(* IEC 61131-3 sources: SmartHomeNew/snapshots/2026-05-07 (part 2) *)

(* ---- FB_Modbus_RTU_SysCom_Backend.st ---- *)
FUNCTION_BLOCK FB_Modbus_RTU_SysCom_Backend
VAR_INPUT
    VI_Enable : BOOL;
    VI_System_Time_MS : UDINT;
END_VAR

VAR
    L_Result : UDINT;
    L_Handle : UDINT := 16#FFFFFFFF;

    L_Settings : SysCom.SysComSettings;
    L_SettingsEx2 : SysCom.SysComSettingsEx2;

    L_Bytes_Written : UDINT;
    L_Bytes_Read : UDINT;

    L_RX_Buffer : ARRAY[0..255] OF BYTE;

    L_Open_Done : BOOL := FALSE;
    L_i : INT;
    L_j : INT;
    L_Read_Count : INT;
    L_Target_Index : INT;
    L_Frame_Length : INT;

    L_CRC : WORD;
    L_CRC_Frame : WORD;

    L_Baudrate : UDINT;
    L_Interframe_MS : UDINT;
END_VAR

// ======================================================
// MODBUS RTU SYSCOM BACKEND
// ======================================================
// Industrial transport runtime:
//   - serial open/configure
//   - RX assembler
//   - CRC validation
//   - watchdog supervision
//   - reconnect supervision
// ======================================================

IF NOT VI_Enable THEN

    IF L_Handle <> 16#FFFFFFFF THEN
        SysCom.SysComClose(hCom := L_Handle);
        L_Handle := 16#FFFFFFFF;
    END_IF;

    L_Open_Done := FALSE;

    GVL_MODBUS_SYSCOM_TRANSPORT.G_Transport_Attached := FALSE;
    GVL_MODBUS_SYSCOM_TRANSPORT.G_Backend_Online := FALSE;

    GVL_MODBUS_SYSCOM_TRANSPORT.G_Backend_State :=
        MB_SYSCOM_CLOSED;

    GVL_MODBUS_SYSCOM_TRANSPORT.G_RX_State :=
        MB_RTU_RX_IDLE;

    GVL_MODBUS_SYSCOM_TRANSPORT.G_RX_Assembler_Active := FALSE;
    GVL_MODBUS_SYSCOM_TRANSPORT.G_RX_Assembler_Length := 0;

    RETURN;
END_IF;

// ======================================================
// WATCHDOGS
// ======================================================
GVL_MODBUS_SYSCOM_TRANSPORT.G_TX_Watchdog_Timeout := FALSE;
GVL_MODBUS_SYSCOM_TRANSPORT.G_RX_Watchdog_Timeout := FALSE;
GVL_MODBUS_SYSCOM_TRANSPORT.G_Bus_Silent := FALSE;

IF GVL_MODBUS_SYSCOM_TRANSPORT.G_TX_Request THEN

    IF (VI_System_Time_MS -
        GVL_MODBUS_SYSCOM_TRANSPORT.G_Last_TX_Request_MS) >
        (GVL_CONFIG.G_Modbus_RTU_Request_Timeout_MS * 2) THEN

        GVL_MODBUS_SYSCOM_TRANSPORT.G_TX_Watchdog_Timeout := TRUE;

        GVL_MODBUS_SYSCOM_TRANSPORT.G_Total_TX_Watchdog :=
            GVL_MODBUS_SYSCOM_TRANSPORT.G_Total_TX_Watchdog + 1;

    END_IF;

END_IF;

IF GVL_MODBUS_SYSCOM_TRANSPORT.G_Backend_Online THEN

    IF (VI_System_Time_MS -
        GVL_MODBUS_SYSCOM_TRANSPORT.G_Last_RX_MS) > 30000 THEN

        GVL_MODBUS_SYSCOM_TRANSPORT.G_RX_Watchdog_Timeout := TRUE;

        GVL_MODBUS_SYSCOM_TRANSPORT.G_Total_RX_Watchdog :=
            GVL_MODBUS_SYSCOM_TRANSPORT.G_Total_RX_Watchdog + 1;

        GVL_MODBUS_SYSCOM_TRANSPORT.G_Bus_Silent := TRUE;

    END_IF;

END_IF;

// ======================================================
// RECONNECT WAIT STATE
// ======================================================
IF GVL_MODBUS_SYSCOM_TRANSPORT.G_Backend_State =
   MB_SYSCOM_RECONNECT_WAIT THEN

    IF (VI_System_Time_MS -
        GVL_MODBUS_SYSCOM_TRANSPORT.G_Backend_Last_Error_MS) >=
        GVL_MODBUS_SYSCOM_TRANSPORT.G_Backend_Reconnect_Delay_MS THEN

        GVL_MODBUS_SYSCOM_TRANSPORT.G_Backend_State :=
            MB_SYSCOM_OPENING;

    ELSE

        RETURN;

    END_IF;

END_IF;

// ======================================================
// OPEN + CONFIGURE
// ======================================================
IF NOT L_Open_Done THEN

    GVL_MODBUS_SYSCOM_TRANSPORT.G_Backend_State :=
        MB_SYSCOM_OPENING;

    L_Baudrate := GVL_CONFIG.G_Modbus_RTU_Baudrate;

    IF L_Baudrate <= 9600 THEN
        L_Interframe_MS := 5;
    ELSIF L_Baudrate <= 19200 THEN
        L_Interframe_MS := 3;
    ELSE
        L_Interframe_MS := 2;
    END_IF;

    GVL_MODBUS_SYSCOM_TRANSPORT.G_RX_Assembler_InterFrame_MS :=
        L_Interframe_MS;

    CASE GVL_CONFIG.G_Modbus_RTU_Port_Number OF
        1:
            L_Settings.sPort := SysCom.SYS_COMPORT1;
        2:
            L_Settings.sPort := SysCom.SYS_COMPORT2;
        3:
            L_Settings.sPort := SysCom.SYS_COMPORT3;
        4:
            L_Settings.sPort := SysCom.SYS_COMPORT4;
    ELSE
        L_Settings.sPort := SysCom.SYS_COMPORT1;
    END_CASE;

    CASE GVL_CONFIG.G_Modbus_RTU_Baudrate OF
        4800:
            L_Settings.ulBaudrate := SysCom.SYS_BR_4800;
        9600:
            L_Settings.ulBaudrate := SysCom.SYS_BR_9600;
        19200:
            L_Settings.ulBaudrate := SysCom.SYS_BR_19200;
        38400:
            L_Settings.ulBaudrate := SysCom.SYS_BR_38400;
        57600:
            L_Settings.ulBaudrate := SysCom.SYS_BR_57600;
        115200:
            L_Settings.ulBaudrate := SysCom.SYS_BR_115200;
    ELSE
        L_Settings.ulBaudrate := SysCom.SYS_BR_9600;
    END_CASE;

    CASE GVL_CONFIG.G_Modbus_RTU_Parity OF
        0:
            L_Settings.byParity := SysCom.SYS_NOPARITY;
        1:
            L_Settings.byParity := SysCom.SYS_EVENPARITY;
        2:
            L_Settings.byParity := SysCom.SYS_ODDPARITY;
    ELSE
        L_Settings.byParity := SysCom.SYS_EVENPARITY;
    END_CASE;

    CASE GVL_CONFIG.G_Modbus_RTU_Stop_Bits OF
        1:
            L_Settings.byStopBits := SysCom.SYS_ONESTOPBIT;
        2:
            L_Settings.byStopBits := SysCom.SYS_TWOSTOPBITS;
    ELSE
        L_Settings.byStopBits := SysCom.SYS_ONESTOPBIT;
    END_CASE;

    L_Settings.ulTimeout := GVL_CONFIG.G_Modbus_RTU_Request_Timeout_MS;
    L_Settings.ulBufferSize := 512;

    IF GVL_CONFIG.G_Modbus_RTU_Data_Bits < 7 THEN
        L_SettingsEx2.byByteSize := 8;
    ELSIF GVL_CONFIG.G_Modbus_RTU_Data_Bits > 8 THEN
        L_SettingsEx2.byByteSize := 8;
    ELSE
        L_SettingsEx2.byByteSize := GVL_CONFIG.G_Modbus_RTU_Data_Bits;
    END_IF;

    L_SettingsEx2.bBinary := TRUE;
    L_SettingsEx2.bOutxCtsFlow := FALSE;
    L_SettingsEx2.bOutxDsrFlow := FALSE;
    L_SettingsEx2.byDtrControl := 0;
    L_SettingsEx2.bDsrSensitivity := FALSE;
    L_SettingsEx2.byRtsControl := 0;
    L_SettingsEx2.bTXContinueOnXoff := FALSE;
    L_SettingsEx2.bOutX := FALSE;
    L_SettingsEx2.bInX := FALSE;
    L_SettingsEx2.byXonChar := 0;
    L_SettingsEx2.byXoffChar := 0;
    L_SettingsEx2.wXonLim := 0;
    L_SettingsEx2.wXoffLim := 0;

    L_Handle := SysCom.SysComOpen3(
        pSettings := ADR(L_Settings),
        pSettingsEx2 := ADR(L_SettingsEx2),
        pResult := ADR(L_Result)
    );

    IF L_Handle <> 16#FFFFFFFF THEN

        SysCom.SysComPurge(hCom := L_Handle);

        L_Open_Done := TRUE;

        GVL_MODBUS_SYSCOM_TRANSPORT.G_Transport_Attached := TRUE;
        GVL_MODBUS_SYSCOM_TRANSPORT.G_Backend_Online := TRUE;

        GVL_MODBUS_SYSCOM_TRANSPORT.G_Backend_State :=
            MB_SYSCOM_ONLINE;

    ELSE

        GVL_MODBUS_SYSCOM_TRANSPORT.G_Transport_Attached := FALSE;
        GVL_MODBUS_SYSCOM_TRANSPORT.G_Backend_Online := FALSE;

        GVL_MODBUS_SYSCOM_TRANSPORT.G_Backend_State :=
            MB_SYSCOM_RECONNECT_WAIT;

        GVL_MODBUS_SYSCOM_TRANSPORT.G_Backend_Last_Error_MS :=
            VI_System_Time_MS;

        GVL_MODBUS_SYSCOM_TRANSPORT.G_Backend_Reconnect_Attempts :=
            GVL_MODBUS_SYSCOM_TRANSPORT.G_Backend_Reconnect_Attempts + 1;

        GVL_MODBUS_SYSCOM_TRANSPORT.G_Total_Reconnects :=
            GVL_MODBUS_SYSCOM_TRANSPORT.G_Total_Reconnects + 1;

        GVL_MODBUS_SYSCOM_TRANSPORT.G_Total_Errors :=
            GVL_MODBUS_SYSCOM_TRANSPORT.G_Total_Errors + 1;

    END_IF;

    RETURN;
END_IF;

GVL_MODBUS_SYSCOM_TRANSPORT.G_Backend_State :=
    MB_SYSCOM_ONLINE;

// ======================================================
// TX WRITE
// ======================================================
IF GVL_MODBUS_SYSCOM_TRANSPORT.G_TX_Request AND
   NOT GVL_MODBUS_SYSCOM_TRANSPORT.G_TX_Done THEN

    L_Bytes_Written := SysCom.SysComWrite(
        hCom := L_Handle,
        pbyBuffer := ADR(GVL_MODBUS_SYSCOM_TRANSPORT.G_TX_Buffer),
        ulSize := GVL_MODBUS_SYSCOM_TRANSPORT.G_TX_Length,
        ulTimeout := GVL_CONFIG.G_Modbus_RTU_Request_Timeout_MS,
        pResult := ADR(L_Result)
    );

    IF L_Bytes_Written = GVL_MODBUS_SYSCOM_TRANSPORT.G_TX_Length THEN

        GVL_MODBUS_SYSCOM_TRANSPORT.G_TX_Done := TRUE;

    ELSE

        GVL_MODBUS_SYSCOM_TRANSPORT.G_TX_Error := TRUE;

        GVL_MODBUS_SYSCOM_TRANSPORT.G_Backend_State :=
            MB_SYSCOM_ERROR;

    END_IF;

END_IF;

// ======================================================
// RX STREAM READ
// ======================================================
L_Bytes_Read := SysCom.SysComRead(
    hCom := L_Handle,
    pbyBuffer := ADR(L_RX_Buffer),
    ulSize := 256,
    ulTimeout := SysCom.SYS_NOWAIT,
    pResult := ADR(L_Result)
);

IF L_Bytes_Read > 0 THEN

    GVL_MODBUS_SYSCOM_TRANSPORT.G_RX_State :=
        MB_RTU_RX_RECEIVING;

    IF L_Bytes_Read > 256 THEN
        L_Read_Count := 256;
    ELSE
        L_Read_Count := UDINT_TO_INT(L_Bytes_Read);
    END_IF;

    GVL_MODBUS_SYSCOM_TRANSPORT.G_RX_Assembler_Active := TRUE;

    GVL_MODBUS_SYSCOM_TRANSPORT.G_RX_Assembler_Last_Byte_MS :=
        VI_System_Time_MS;

    FOR L_i := 0 TO (L_Read_Count - 1) DO

        L_Target_Index :=
            UINT_TO_INT(GVL_MODBUS_SYSCOM_TRANSPORT.G_RX_Assembler_Length);

        IF L_Target_Index >= 256 THEN

            GVL_MODBUS_SYSCOM_TRANSPORT.G_RX_State :=
                MB_RTU_RX_OVERFLOW;

            GVL_MODBUS_SYSCOM_TRANSPORT.G_RX_Assembler_Overflow := TRUE;

            GVL_MODBUS_SYSCOM_TRANSPORT.G_Total_RX_Overflow :=
                GVL_MODBUS_SYSCOM_TRANSPORT.G_Total_RX_Overflow + 1;

            GVL_MODBUS_SYSCOM_TRANSPORT.G_RX_Assembler_Active := FALSE;
            GVL_MODBUS_SYSCOM_TRANSPORT.G_RX_Assembler_Length := 0;

            EXIT;

        END_IF;

        GVL_MODBUS_SYSCOM_TRANSPORT.G_RX_Buffer[L_Target_Index] :=
            L_RX_Buffer[L_i];

        GVL_MODBUS_SYSCOM_TRANSPORT.G_RX_Assembler_Length :=
            GVL_MODBUS_SYSCOM_TRANSPORT.G_RX_Assembler_Length + 1;

    END_FOR;

END_IF;

// ======================================================
// INTER-FRAME FINALIZATION
// ======================================================
IF GVL_MODBUS_SYSCOM_TRANSPORT.G_RX_Assembler_Active THEN

    IF (VI_System_Time_MS -
        GVL_MODBUS_SYSCOM_TRANSPORT.G_RX_Assembler_Last_Byte_MS) >=
        GVL_MODBUS_SYSCOM_TRANSPORT.G_RX_Assembler_InterFrame_MS THEN

        L_Frame_Length :=
            UINT_TO_INT(GVL_MODBUS_SYSCOM_TRANSPORT.G_RX_Assembler_Length);

        IF L_Frame_Length >= 4 THEN

            L_CRC := 16#FFFF;

            FOR L_i := 0 TO (L_Frame_Length - 3) DO

                L_CRC := L_CRC XOR
                    BYTE_TO_WORD(
                        GVL_MODBUS_SYSCOM_TRANSPORT.G_RX_Buffer[L_i]
                    );

                FOR L_j := 0 TO 7 DO

                    IF (L_CRC AND 16#0001) <> 0 THEN
                        L_CRC := SHR(L_CRC, 1);
                        L_CRC := L_CRC XOR 16#A001;
                    ELSE
                        L_CRC := SHR(L_CRC, 1);
                    END_IF;

                END_FOR;

            END_FOR;

            L_CRC_Frame :=
                BYTE_TO_WORD(
                    GVL_MODBUS_SYSCOM_TRANSPORT.G_RX_Buffer[L_Frame_Length - 2]
                );

            L_CRC_Frame :=
                L_CRC_Frame OR
                SHL(
                    BYTE_TO_WORD(
                        GVL_MODBUS_SYSCOM_TRANSPORT.G_RX_Buffer[L_Frame_Length - 1]
                    ),
                    8
                );

            GVL_MODBUS_SYSCOM_TRANSPORT.G_RX_Assembler_CRC_Calc :=
                L_CRC;

            GVL_MODBUS_SYSCOM_TRANSPORT.G_RX_Assembler_CRC_Frame :=
                L_CRC_Frame;

            IF L_CRC = L_CRC_Frame THEN

                GVL_MODBUS_SYSCOM_TRANSPORT.G_RX_State :=
                    MB_RTU_RX_FRAME_READY;

                GVL_MODBUS_SYSCOM_TRANSPORT.G_RX_Assembler_CRC_OK := TRUE;

                GVL_MODBUS_SYSCOM_TRANSPORT.G_RX_Length :=
                    GVL_MODBUS_SYSCOM_TRANSPORT.G_RX_Assembler_Length;

                GVL_MODBUS_SYSCOM_TRANSPORT.G_RX_Ready := TRUE;

                GVL_MODBUS_SYSCOM_TRANSPORT.G_Total_RX :=
                    GVL_MODBUS_SYSCOM_TRANSPORT.G_Total_RX + 1;

                GVL_MODBUS_SYSCOM_TRANSPORT.G_Last_RX_MS :=
                    VI_System_Time_MS;

            ELSE

                GVL_MODBUS_SYSCOM_TRANSPORT.G_RX_State :=
                    MB_RTU_RX_CRC_ERROR;

                GVL_MODBUS_SYSCOM_TRANSPORT.G_RX_Assembler_CRC_OK := FALSE;

                GVL_MODBUS_SYSCOM_TRANSPORT.G_Total_RX_CRC_Error :=
                    GVL_MODBUS_SYSCOM_TRANSPORT.G_Total_RX_CRC_Error + 1;

            END_IF;

        ELSE

            GVL_MODBUS_SYSCOM_TRANSPORT.G_RX_State :=
                MB_RTU_RX_SHORT_FRAME;

            GVL_MODBUS_SYSCOM_TRANSPORT.G_Total_RX_Short_Frame :=
                GVL_MODBUS_SYSCOM_TRANSPORT.G_Total_RX_Short_Frame + 1;

        END_IF;

        GVL_MODBUS_SYSCOM_TRANSPORT.G_RX_Assembler_Active := FALSE;
        GVL_MODBUS_SYSCOM_TRANSPORT.G_RX_Assembler_Length := 0;

    END_IF;

END_IF;

IF NOT GVL_MODBUS_SYSCOM_TRANSPORT.G_RX_Assembler_Active AND
   NOT GVL_MODBUS_SYSCOM_TRANSPORT.G_RX_Ready AND
   (GVL_MODBUS_SYSCOM_TRANSPORT.G_RX_State = MB_RTU_RX_FRAME_READY) THEN

    GVL_MODBUS_SYSCOM_TRANSPORT.G_RX_State :=
        MB_RTU_RX_IDLE;

END_IF;

END_FUNCTION_BLOCK

(* ---- FB_System_Diagnostics.st ---- *)
// ==============================================================================
// System diagnostics helper
//
// Internal helper for PRG_System.
// Owns diagnostic flag export into GVL_STATUS.G_Diagnostics.
// ==============================================================================
FUNCTION_BLOCK FB_System_Diagnostics

GVL_STATUS.G_Diagnostics.Sensor_Fault :=
    GVL_STATE.G_Heating_Sensor_Fault OR
    GVL_STATE.G_DHW_Sensor_Fault OR
    GVL_STATUS.G_Diagnostics.Manifold_Pressure_Fault_Active OR
    GVL_STATUS.G_Diagnostics.Manifold_Current_Fault_Active OR
    GVL_STATUS.G_Diagnostics.Manifold_Return_Temp_Fault_Active;

GVL_STATUS.G_Diagnostics.IO_Offline :=
    GVL_STATE.G_Heating_IO_Fault OR
    GVL_STATE.G_DHW_IO_Fault OR
    GVL_STATE.G_Ventilation_IO_Fault OR
    GVL_STATE.G_Lighting_IO_Fault;

GVL_STATUS.G_Diagnostics.Subsystem_Degraded :=
    GVL_STATE.G_Heating_Subsystem_Degraded OR
    GVL_STATE.G_DHW_Subsystem_Degraded OR
    GVL_STATE.G_Ventilation_Subsystem_Degraded OR
    GVL_STATUS.G_Diagnostics.Manifold_Pressure_Fault_Active OR
    GVL_STATUS.G_Diagnostics.Manifold_Current_Fault_Active OR
    GVL_STATUS.G_Diagnostics.Manifold_Return_Temp_Fault_Active;

// >>> BULK_SYNC_ANCHOR: FB_System_Diagnostics <<<
END_FUNCTION_BLOCK

(* ---- FB_System_Redundancy_Orchestrator.st ---- *)
// ==============================================================================
// System redundancy orchestrator helper
//
// Internal helper for PRG_System.
// Owns PLC role calculation, heartbeat output projection, and synced-state apply.
// ==============================================================================
FUNCTION_BLOCK FB_System_Redundancy_Orchestrator
VAR_IN_OUT
    VIO_Local_State : ST_System_State_Snapshot;
    VIO_Remote_State : ST_System_State_Snapshot;
END_VAR

VAR
    fbRedundancy : FB_Redundancy_Manager;
END_VAR

// Build local state snapshot for replication.
VIO_Local_State.System_Time_MS := GVL_STATUS.G_System_Time_MS;
VIO_Local_State.Current_Scenario := GVL_STATUS.G_Current_Scenario;
VIO_Local_State.Security_Armed := GVL_ALARM.G_Security_Armed;
VIO_Local_State.Active_Alarms := GVL_ALARM.G_Active_Alarm_Count;
VIO_Local_State.Zone_Valves := GVL_STATE.G_Zone_Valves;
VIO_Local_State.Manifold_Pumps := GVL_STATE.G_Manifold_Pumps;
VIO_Local_State.Lighting_States := GVL_STATE.G_Lighting_Levels;
VIO_Local_State.Blinds_Positions := GVL_STATE.G_Blinds_Positions;
VIO_Local_State.Socket_States := GVL_STATE.G_Socket_States;
VIO_Local_State.Gas_Valve_Closed := GVL_COMMAND.G_Gas_Valve_Close;
VIO_Local_State.Water_Valves_Closed := GVL_COMMAND.G_Close_Valve_36;
VIO_Local_State.Version := VIO_Local_State.Version + 1;

fbRedundancy(
    VI_System_Time_MS := GVL_STATUS.G_System_Time_MS,
    VI_Local_PLC_ID := GVL_STATUS.G_PLC_ID,
    VI_Remote_Pulse := GVL_IO.DI_Partner_Pulse,
    VI_Remote_Is_Active := GVL_IO.DI_Partner_Active,
    VI_Gateway_Ping_OK := GVL_GATEWAY.G_Gateway_Ping_OK,
    VI_Local_State := VIO_Local_State,
    VI_Remote_State := VIO_Remote_State
);

GVL_STATUS.G_Is_Active_PLC := (fbRedundancy.VO_Local_Role = E_PLC_ROLE.ROLE_ACTIVE);
GVL_IO.DO_Heartbeat_Pulse := fbRedundancy.VO_Local_Pulse;
GVL_IO.DO_Active_Status := GVL_STATUS.G_Is_Active_PLC;

IF fbRedundancy.VO_State_Updated THEN
    GVL_STATUS.G_Current_Scenario := fbRedundancy.VO_Synced_State.Current_Scenario;
    GVL_ALARM.G_Security_Armed := fbRedundancy.VO_Synced_State.Security_Armed;
    GVL_STATE.G_Zone_Valves := fbRedundancy.VO_Synced_State.Zone_Valves;
    GVL_STATE.G_Manifold_Pumps := fbRedundancy.VO_Synced_State.Manifold_Pumps;
    GVL_STATE.G_Lighting_Levels := fbRedundancy.VO_Synced_State.Lighting_States;
    GVL_STATE.G_Blinds_Positions := fbRedundancy.VO_Synced_State.Blinds_Positions;
    GVL_STATE.G_Socket_States := fbRedundancy.VO_Synced_State.Socket_States;
    GVL_COMMAND.G_Gas_Valve_Close := fbRedundancy.VO_Synced_State.Gas_Valve_Closed;
    GVL_COMMAND.G_Close_Valve_36 := fbRedundancy.VO_Synced_State.Water_Valves_Closed;
    VIO_Local_State.Version := fbRedundancy.VO_Synced_State.Version;
END_IF;

// >>> BULK_SYNC_ANCHOR: FB_System_Redundancy_Orchestrator <<<
END_FUNCTION_BLOCK

(* ---- FB_System_Timer_TOF.st ---- *)
// ==============================================================================
// Блок таймера задержки выключения (System Timer TOF)
// Назначение:
// - Замена стандартного TOF для обеспечения точной выдержки времени,
//   независимой от времени цикла ПЛК, с использованием единого системного времени.
// ==============================================================================
FUNCTION_BLOCK FB_System_Timer_TOF
VAR_INPUT
    IN : BOOL; // Вход запуска таймера
    PT : TIME; // Заданное время
    VI_System_Time_MS : UDINT; // Системное время (мс)
END_VAR
VAR_OUTPUT
    Q : BOOL; // Выход: таймер сработал
    ET : TIME; // Прошедшее время
END_VAR
VAR
    L_Start_Time : UDINT;
    L_Running : BOOL;
    L_Prev_IN : BOOL;
END_VAR

IF IN THEN
    Q := TRUE;
    ET := T#0s;
    L_Running := FALSE;
ELSE
    IF L_Prev_IN THEN
        L_Start_Time := VI_System_Time_MS;
        L_Running := TRUE;
        ET := T#0s;
    END_IF;

    IF L_Running THEN
        // Обработка переполнения UDINT (примерно 49 дней)
        ET := TO_TIME((SEL(VI_System_Time_MS >= L_Start_Time, VI_System_Time_MS - L_Start_Time, (4294967295 - L_Start_Time) + VI_System_Time_MS + 1)));

        IF ET >= PT THEN
            Q := FALSE;
            ET := PT;
            L_Running := FALSE;
        ELSE
            Q := TRUE;
        END_IF;
    END_IF;
END_IF;

L_Prev_IN := IN;
END_FUNCTION_BLOCK

(* ---- FB_Ventilation_System_Manager.st ---- *)
FUNCTION_BLOCK FB_Ventilation_System_Manager
VAR_INPUT
    VI_System_Time_MS : UDINT; // Системное время (мс)
    VI_IsActivePLC : BOOL; // Флаг: Данный ПЛК является ведущим
    VI_Outdoor_Temp : REAL; // Уличная температура воздуха (°C)
    VI_Current_Scenario : E_SCENARIO_TYPE; // Текущий глобальный сценарий
    VI_System_Mode : E_System_Operating_Mode; // Агрегированный режим работы системы
    VI_Config : ST_Ventilation_Global_Config; // Конфигурация системы вентиляции
    VI_Fire_Alarm : BOOL; // Сигнал пожарной тревоги
    VI_Gas_Alarm : BOOL; // Сигнал газовой тревоги
    VI_PV3_Boost_Req : BOOL; // Запрос форсирования ПВ-3 от газоанализатора (ТЗ 5.1)
    VI_Supply_100_Req : BOOL; // Запрос 100% притока (ТЗ 6.4)
    VI_Exhaust_100_Req : BOOL; // Запрос 100% вытяжки (ТЗ 6.4)
    VI_Supply_80_Req : BOOL; // Запрос 80% притока (ТЗ 5.4)
    VI_Vent_Stop : BOOL; // Запрос на остановку вентиляции (ТЗ 5.3)
    VI_IO_Modules_Online : ARRAY[1..GVL_CONSTANTS.C_MAX_MODULES] OF BOOL; // Статусы модулей ввода-вывода (только чтение)
END_VAR
VAR_IN_OUT
    VI_Supply_Temps : ARRAY[1..GVL_CONSTANTS.C_MAX_SUPPLY_TEMPS] OF REAL; // Температура приточного воздуха после калорифера
    VI_Room_Temps : ARRAY[1..16] OF REAL; // Температура в помещениях (°C)
    VI_Room_Humidities : ARRAY[1..16] OF REAL; // Влажность в помещениях (%)
    VI_Room_CO2 : ARRAY[1..16] OF REAL; // Уровень CO2 в помещениях (ppm)
    VI_Wet_Zone_Active : ARRAY[1..GVL_CONSTANTS.C_MAX_WET_ZONES] OF BOOL; // Сигналы включения света в санузлах (ТЗ 4.0)
    VI_Rule_Actions : ARRAY[1..GVL_CONSTANTS.C_MAX_RULES] OF ST_Rule_Action; // Действия от Rule Engine
END_VAR
VAR_OUTPUT
    VO_Supply_Fans : ARRAY[1..GVL_CONSTANTS.C_MAX_SUPPLY_FANS] OF BYTE; // Выход: Управление приточными вентиляторами (0-100%)
    VO_Exhaust_Fans : ARRAY[1..GVL_CONSTANTS.C_MAX_EXHAUST_FANS] OF BYTE; // Выход: Управление вытяжными вентиляторами (0-100%)
    VO_Heater_Power : ARRAY[1..GVL_CONSTANTS.C_MAX_BOILERS] OF REAL; // Выход: Мощность калориферов (0-100%)
    VO_Status_Msg : STRING(200); // Строковое сообщение о статусе
    VO_Ventilation_IO_Fault : BOOL; // Выход: диагностика потери связи с модулями ввода-вывода
    VO_Ventilation_Subsystem_Degraded : BOOL; // Выход: признак degraded-состояния подсистемы вентиляции
END_VAR
VAR
    L_Policy_Normal : BOOL;
    L_Policy_Safe_Stop : BOOL;
    L_Policy_Degraded : BOOL;
    L_Policy_Freeze_Protection : BOOL;
    L_i : INT;
    L_j : INT;
    L_Max_CO2 : REAL;
    L_Max_Hum : REAL;
    L_Base_Speed : BYTE;
    L_Target_Temp : REAL;
    L_PID_Heaters : ARRAY[1..GVL_CONSTANTS.C_MAX_BOILERS] OF FB_PID_Controller;
    L_Wet_Zone_Timers : ARRAY[1..GVL_CONSTANTS.C_MAX_WET_ZONES] OF FB_System_Timer_TOF; // Таймеры выбега для вытяжек санузлов
END_VAR

// ========================================
// Ventilation policy layer
// ========================================
VO_Ventilation_IO_Fault := FALSE;
VO_Ventilation_Subsystem_Degraded := FALSE;
L_Policy_Normal := (VI_System_Mode = E_System_Operating_Mode.MODE_NORMAL);
L_Policy_Safe_Stop := (VI_System_Mode = E_System_Operating_Mode.MODE_SAFE_STOP);
L_Policy_Degraded := (VI_System_Mode = E_System_Operating_Mode.MODE_DEGRADED);
L_Policy_Freeze_Protection := (VI_System_Mode = E_System_Operating_Mode.MODE_FREEZE_PROTECTION);

IF NOT VI_IsActivePLC THEN
    FOR L_i := 1 TO GVL_CONSTANTS.C_MAX_SUPPLY_FANS DO
        VO_Supply_Fans[L_i] := 0;
        IF L_i <= GVL_CONSTANTS.C_MAX_SUPPLY_TEMPS THEN
            VO_Heater_Power[L_i] := 0.0;
        END_IF;
    END_FOR;
    FOR L_i := 1 TO GVL_CONSTANTS.C_MAX_EXHAUST_FANS DO
        VO_Exhaust_Fans[L_i] := 0;
    END_FOR;
    VO_Status_Msg := 'ВЕНТИЛЯЦИЯ: РЕЗЕРВНЫЙ ПЛК';
    RETURN;
END_IF;

// Проверка связи с модулями ввода-вывода
FOR L_i := 1 TO GVL_CONSTANTS.C_MAX_MODULES DO
    IF NOT VI_IO_Modules_Online[L_i] THEN
        VO_Ventilation_IO_Fault := TRUE;
        FOR L_j := 1 TO GVL_CONSTANTS.C_MAX_SUPPLY_FANS DO
            VO_Supply_Fans[L_j] := 0;
        END_FOR;
        FOR L_j := 1 TO GVL_CONSTANTS.C_MAX_EXHAUST_FANS DO
            VO_Exhaust_Fans[L_j] := 0;
        END_FOR;
        FOR L_j := 1 TO GVL_CONSTANTS.C_MAX_BOILERS DO
            VO_Heater_Power[L_j] := 0.0;
        END_FOR;
        VO_Status_Msg := 'ОШИБКА: Потеря связи с модулями ввода-вывода';
        RETURN;
    END_IF;
END_FOR;

// =========================
// SYSTEM MODE / HARD REQUEST OVERRIDES
// =========================
IF L_Policy_Safe_Stop OR VI_Vent_Stop THEN
    FOR L_i := 1 TO GVL_CONSTANTS.C_MAX_SUPPLY_FANS DO
        VO_Supply_Fans[L_i] := 0;
    END_FOR;
    FOR L_i := 1 TO GVL_CONSTANTS.C_MAX_EXHAUST_FANS DO
        VO_Exhaust_Fans[L_i] := 0;
    END_FOR;
    FOR L_i := 1 TO GVL_CONSTANTS.C_MAX_BOILERS DO
        VO_Heater_Power[L_i] := 0.0;
    END_FOR;
    IF VI_Vent_Stop THEN
        VO_Status_Msg := 'ВЕНТИЛЯЦИЯ: ОСТАНОВЛЕНА ПО КОМАНДЕ';
    ELSE
        VO_Status_Msg := 'ВЕНТИЛЯЦИЯ: ОСТАНОВЛЕНА POLICY SAFE_STOP';
    END_IF;
    RETURN;
END_IF;

IF L_Policy_Degraded THEN
    FOR L_i := 1 TO GVL_CONSTANTS.C_MAX_SUPPLY_FANS DO
        VO_Supply_Fans[L_i] := 0;
    END_FOR;
    FOR L_i := 1 TO GVL_CONSTANTS.C_MAX_BOILERS DO
        VO_Heater_Power[L_i] := 0.0;
    END_FOR;
    VO_Ventilation_Subsystem_Degraded := TRUE;
    VO_Status_Msg := 'ВЕНТИЛЯЦИЯ: DEGRADED POLICY';
END_IF;

IF L_Policy_Freeze_Protection THEN
    FOR L_i := 1 TO GVL_CONSTANTS.C_MAX_SUPPLY_FANS DO
        VO_Supply_Fans[L_i] := 0;
    END_FOR;
    FOR L_i := 1 TO GVL_CONSTANTS.C_MAX_EXHAUST_FANS DO
        VO_Exhaust_Fans[L_i] := 0;
    END_FOR;
    FOR L_i := 1 TO GVL_CONSTANTS.C_MAX_BOILERS DO
        VO_Heater_Power[L_i] := 0.0;
    END_FOR;
    VO_Status_Msg := 'ВЕНТИЛЯЦИЯ: FREEZE_PROTECTION POLICY (stop)';
    RETURN;
END_IF;

// 1. Определение базовой скорости и целевой температуры по сценарию (ТЗ 7.1)
CASE VI_Current_Scenario OF
    E_SCENARIO_TYPE.SCENARIO_AWAY:
        L_Base_Speed := VI_Config.Scenario_Modes[3].Base_Fan_Speed;
        L_Target_Temp := VI_Config.Scenario_Modes[3].Target_Temp;
    E_SCENARIO_TYPE.SCENARIO_SLEEP:
        L_Base_Speed := VI_Config.Scenario_Modes[2].Base_Fan_Speed;
        L_Target_Temp := VI_Config.Scenario_Modes[2].Target_Temp;
    ELSE // PRESENCE, MORNING, EVENING
        L_Base_Speed := VI_Config.Scenario_Modes[1].Base_Fan_Speed;
        L_Target_Temp := VI_Config.Scenario_Modes[1].Target_Temp;
END_CASE;

// 2. Логика управления приточными установками (П-1, П-2, П-3)
FOR L_i := 1 TO GVL_CONSTANTS.C_MAX_SUPPLY_FANS DO
    IF L_i <= GVL_CONSTANTS.C_MAX_SUPPLY_TEMPS THEN
        L_PID_Heaters[L_i](
            VI_SetPoint := L_Target_Temp,
            VI_ProcessValue := VI_Supply_Temps[L_i],
            VI_Kp := 4.0, VI_Tn := 120.0, VI_Tv := 0.0,
            VI_Y_Min := 0.0, VI_Y_Max := 100.0, VI_Cycle_Time_S := 1.0,
            VO_Output => VO_Heater_Power[L_i]
        );
    END_IF;

    VO_Supply_Fans[L_i] := L_Base_Speed;

    FOR L_j := 1 TO GVL_CONSTANTS.C_MAX_RULES DO
        IF VI_Rule_Actions[L_j].Active AND VI_Rule_Actions[L_j].Target_ID = L_i THEN
            IF VI_Rule_Actions[L_j].Action_Type = E_Rule_Action_Type.ACTION_SET_VENTILATION THEN
                VO_Supply_Fans[L_i] := REAL_TO_BYTE(VI_Rule_Actions[L_j].Value);
            END_IF;
        END_IF;
    END_FOR;
END_FOR;

// 3. Логика управления вытяжными установками (В-1 .. В-5)
FOR L_i := 1 TO GVL_CONSTANTS.C_MAX_EXHAUST_FANS DO
    VO_Exhaust_Fans[L_i] := L_Base_Speed;

    FOR L_j := 1 TO GVL_CONSTANTS.C_MAX_WET_ZONES DO
        IF VI_Config.wet_zone_to_exhaust_map[L_j] = L_i THEN
            L_Wet_Zone_Timers[L_j](IN := VI_Wet_Zone_Active[L_j], PT := T#5m, VI_System_Time_MS := VI_System_Time_MS);
            IF VI_Wet_Zone_Active[L_j] THEN
                VO_Exhaust_Fans[L_i] := 80;
            ELSIF L_Wet_Zone_Timers[L_j].Q THEN
                VO_Exhaust_Fans[L_i] := 50;
            END_IF;
        END_IF;
    END_FOR;
END_FOR;

// ========================================
// OPERATIONAL REQUEST OVERRIDES
// ========================================
IF VI_Supply_100_Req THEN
    FOR L_i := 1 TO GVL_CONSTANTS.C_MAX_SUPPLY_FANS DO
        VO_Supply_Fans[L_i] := 100;
    END_FOR;
ELSIF VI_Supply_80_Req THEN
    FOR L_i := 1 TO GVL_CONSTANTS.C_MAX_SUPPLY_FANS DO
        IF VO_Supply_Fans[L_i] < 80 THEN
            VO_Supply_Fans[L_i] := 80;
        END_IF;
    END_FOR;
END_IF;

IF VI_PV3_Boost_Req THEN
    IF GVL_CONSTANTS.C_MAX_SUPPLY_FANS >= 3 THEN
        VO_Supply_Fans[3] := 100;
    END_IF;
END_IF;

IF VI_Exhaust_100_Req THEN
    FOR L_i := 1 TO GVL_CONSTANTS.C_MAX_EXHAUST_FANS DO
        VO_Exhaust_Fans[L_i] := 100;
    END_FOR;
END_IF;

// ========================================
// VENT_FINAL_CLAMP
// ========================================
IF L_Policy_Degraded THEN
    FOR L_i := 1 TO GVL_CONSTANTS.C_MAX_EXHAUST_FANS DO
        VO_Exhaust_Fans[L_i] := MIN(VO_Exhaust_Fans[L_i], VI_Config.Degraded_Exhaust_Limit);
    END_FOR;
END_IF;

// 4. Формирование статусного сообщения
IF L_Policy_Degraded THEN
    VO_Status_Msg := 'ВЕНТИЛЯЦИЯ: DEGRADED POLICY';
ELSIF VI_PV3_Boost_Req OR VI_Supply_100_Req OR VI_Exhaust_100_Req OR VI_Supply_80_Req THEN
    VO_Status_Msg := 'Вентиляция: активен операционный boost/request';
ELSE
    VO_Status_Msg := 'Вентиляция работает в штатном режиме';
END_IF;
// >>> BULK_SYNC_ANCHOR: FB_Ventilation_System_Manager <<<
END_FUNCTION_BLOCK

(* ---- MAIN.st ---- *)
PROGRAM MAIN

// ======================================================
// MAIN CYCLIC EXECUTION PIPELINE
// ======================================================
// Required CODESYS Task Configuration:
//   - Assign only PROGRAM MAIN to the cyclic task.
//   - Do not assign child PRG_* programs directly to the same task.
//   - Configure the real cycle time in CODESYS Task Configuration.
//   - Recommended main control cycle: 100 ms.
//
// Execution principle:
//   1. Time / init / configuration
//   2. PLC role arbitration
//   3. IO read and input normalization
//   4. Mode, presence and safety
//   5. Intent, behavior, scenario and policy
//   6. Command arbitration
//   7. Domain execution
//   8. Physical IO write
//   9. Verification, diagnostics, history, HMI
// ======================================================

// 1. Time / init / configuration
PRG_Time_Service();
PRG_System_Init();
PRG_Config_Manager();
PRG_Config_Validation();
PRG_Config_Versioning();
PRG_System_Runtime_Base();

// 2. PLC role arbitration
PRG_PLC_Arbitration();

// 3. IO read and normalized inputs
PRG_IO_Read();
PRG_Input_Processing();

// 4. Base mode, presence and safety
PRG_Mode_Manager();
PRG_Presence_Manager();
PRG_Safety();
PRG_Safety_Operator();
PRG_Safety_Shutdown();
PRG_Safety_Recovery();

// 5. Intent, adaptive behavior, scenario and policy
PRG_System_Intent();
PRG_Security();
PRG_System_Access_Maintenance();
PRG_User_Adapt_Control();
PRG_Behavior_Adapt_Profile();
PRG_Scenario_Engine();
PRG_System_Scenario_Rules();
PRG_System_Evacuation();
PRG_Policy();
PRG_Heating_Policy_Manager();
PRG_Heating_Policy_Observer();
PRG_System_Coordinator();

// 6. Command arbitration
PRG_Command_Arbitration();

// 6.5 Modbus/OpenTherm transport pipeline.
// Modbus master schedules requests.
// RTU bridge exports request/imports confirmed response.
// RTU driver builds TX frame and consumes validated RX frame.
// SysCom backend performs physical serial IO.
// SysCom transport boundary transfers bytes between backend and RTU runtime.
// Register scanner is strictly read-only diagnostics.
// OpenTherm transport decodes wire image before validation.
PRG_Modbus_Master();
PRG_Modbus_RTU_Bridge();
PRG_Modbus_RTU_Driver();
PRG_Modbus_RTU_SysCom_Backend();
PRG_Modbus_RTU_SysCom_Transport();
PRG_Modbus_Register_Scan();
PRG_OpenTherm_Transport();
PRG_OpenTherm_Adapter_Status();

// 7. Domain execution and domain output projection
PRG_Heating();
PRG_Ventilation();
PRG_Water();
PRG_Access();
PRG_Lighting();

// 8. Final physical IO projection. Must remain after all domain execution.
PRG_IO_Write();

// 9. Verification, explainability, diagnostics, history, HMI
PRG_Command_Verifier();
PRG_Explainability();
PRG_System_Health();
PRG_System_Alarm_Gateway();
PRG_System_Diagnostics();
PRG_System_Diagnostics_Ext();
PRG_System_History();
PRG_System_BlackBox();
PRG_System_Trend();
PRG_System_Simulation();
PRG_HMI_Dashboard();
PRG_Debug_View();

// >>> BULK_SYNC_ANCHOR: MAIN <<<
END_PROGRAM

(* ---- PRG_Behavior_Adapt_Profile.st ---- *)
PROGRAM PRG_Behavior_Adapt_Profile

// Centralized tuning profile controller.
// This block enforces consistent adaptive behavior settings.

CASE GVL_BEHAVIOR_ADAPT.G_Adapt_Profile OF

    ADAPT_PROFILE_STABLE:
        GVL_BEHAVIOR_ADAPT.G_Adapt_Learning_Rate := 0.03;
        GVL_BEHAVIOR_ADAPT.G_Confidence_Learning_Rate := 0.03;
        GVL_BEHAVIOR_ADAPT.G_Decay_Factor := 0.998;
        GVL_BEHAVIOR_ADAPT.G_Adapt_Update_Threshold := 7;

        GVL_BEHAVIOR_ADAPT.G_Behavior_Weight_Comfort := 1.0;
        GVL_BEHAVIOR_ADAPT.G_Behavior_Weight_Night := 1.0;
        GVL_BEHAVIOR_ADAPT.G_Behavior_Weight_Preheat := 1.0;
        GVL_BEHAVIOR_ADAPT.G_Behavior_Weight_VentBoost := 0.9;
        GVL_BEHAVIOR_ADAPT.G_Behavior_Weight_AccessSecure := 1.0;

    ADAPT_PROFILE_BALANCED:
        GVL_BEHAVIOR_ADAPT.G_Adapt_Learning_Rate := 0.05;
        GVL_BEHAVIOR_ADAPT.G_Confidence_Learning_Rate := 0.05;
        GVL_BEHAVIOR_ADAPT.G_Decay_Factor := 0.995;
        GVL_BEHAVIOR_ADAPT.G_Adapt_Update_Threshold := 5;

        GVL_BEHAVIOR_ADAPT.G_Behavior_Weight_Comfort := 1.0;
        GVL_BEHAVIOR_ADAPT.G_Behavior_Weight_Night := 1.0;
        GVL_BEHAVIOR_ADAPT.G_Behavior_Weight_Preheat := 1.0;
        GVL_BEHAVIOR_ADAPT.G_Behavior_Weight_VentBoost := 1.0;
        GVL_BEHAVIOR_ADAPT.G_Behavior_Weight_AccessSecure := 1.0;

    ADAPT_PROFILE_AGGRESSIVE:
        GVL_BEHAVIOR_ADAPT.G_Adapt_Learning_Rate := 0.08;
        GVL_BEHAVIOR_ADAPT.G_Confidence_Learning_Rate := 0.08;
        GVL_BEHAVIOR_ADAPT.G_Decay_Factor := 0.990;
        GVL_BEHAVIOR_ADAPT.G_Adapt_Update_Threshold := 3;

        GVL_BEHAVIOR_ADAPT.G_Behavior_Weight_Comfort := 1.0;
        GVL_BEHAVIOR_ADAPT.G_Behavior_Weight_Night := 1.0;
        GVL_BEHAVIOR_ADAPT.G_Behavior_Weight_Preheat := 1.0;
        GVL_BEHAVIOR_ADAPT.G_Behavior_Weight_VentBoost := 1.1;
        GVL_BEHAVIOR_ADAPT.G_Behavior_Weight_AccessSecure := 1.0;

ELSE
        // No fallback required
END_CASE;

// >>> BULK_SYNC_ANCHOR: PRG_Behavior_Adapt_Profile <<<
END_PROGRAM

(* ---- PRG_Config_Simulation.st ---- *)
PROGRAM PRG_Config_Simulation
VAR
    L_Error : BOOL;
END_VAR

L_Error := FALSE;
GVL_CONFIG_SIMULATION.G_Simulation_Result_OK := TRUE;
GVL_CONFIG_SIMULATION.G_Simulation_Error_Text := '';

IF GVL_CONFIG_SIMULATION.G_Simulation_Request AND GVL_CONFIG_SIMULATION.G_Simulation_Confirm THEN

    // Simulate INPUT constraints
    IF (GVL_CONFIG_CONTROL.STG_Reputation_Learning_Rate < 0.0) OR (GVL_CONFIG_CONTROL.STG_Reputation_Learning_Rate > 1.0) THEN
        GVL_CONFIG_SIMULATION.G_Simulation_Result_OK := FALSE;
        GVL_CONFIG_SIMULATION.G_Simulation_Error_Text := 'Invalid learning rate';
        L_Error := TRUE;
    END_IF;

    // Simulate SCENARIO logic
    IF GVL_CONFIG_CONTROL.STG_Night_Start_Hour = GVL_CONFIG_CONTROL.STG_Night_End_Hour THEN
        GVL_CONFIG_SIMULATION.G_Simulation_Result_OK := FALSE;
        GVL_CONFIG_SIMULATION.G_Simulation_Error_Text := 'Night window invalid';
        L_Error := TRUE;
    END_IF;

    // Simulate SAFETY
    IF GVL_CONFIG_CONTROL.STG_Stabilization_Delay_MS < 1000 THEN
        GVL_CONFIG_SIMULATION.G_Simulation_Result_OK := FALSE;
        GVL_CONFIG_SIMULATION.G_Simulation_Error_Text := 'Recovery delay too small';
        L_Error := TRUE;
    END_IF;

    // Simulate FAIL-SAFE policy
    IF NOT (
        GVL_CONFIG_CONTROL.STG_PLC_Inactive_Close_Gas OR
        GVL_CONFIG_CONTROL.STG_PLC_Inactive_Stop_Boiler OR
        GVL_CONFIG_CONTROL.STG_PLC_Inactive_Block_Heating OR
        GVL_CONFIG_CONTROL.STG_PLC_Inactive_Stop_Vent OR
        GVL_CONFIG_CONTROL.STG_PLC_Inactive_Block_Water
    ) THEN
        GVL_CONFIG_SIMULATION.G_Simulation_Result_OK := FALSE;
        GVL_CONFIG_SIMULATION.G_Simulation_Error_Text := 'Fail-safe disabled';
        L_Error := TRUE;
    END_IF;

    GVL_CONFIG_SIMULATION.G_Simulation_Last_Run_MS := GVL_TIME_SERVICE.G_Now_MS;

END_IF;

// >>> BULK_SYNC_ANCHOR: PRG_Config_Simulation <<<
END_PROGRAM

(* ---- PRG_HMI_Dashboard.st ---- *)
PROGRAM PRG_HMI_Dashboard
VAR
    L_i : INT;
END_VAR

// ======================================================
// HEATING CONFIDENCE
// ======================================================
GVL_HMI.G_HMI_Heating_Confidence := GVL_STATE.G_Heating_Confidence;
GVL_HMI.G_HMI_Heating_Confidence_Percent := REAL_TO_INT(GVL_STATE.G_Heating_Confidence * 100.0);

// ======================================================
// HEATING ROOT CAUSE
// ======================================================
GVL_HMI.G_HMI_Heating_Reason_Code := GVL_STATE.G_Heating_Confidence_Reason_Code;
GVL_HMI.G_HMI_Heating_Status_Text := GVL_STATE.G_Heating_Confidence_Reason_Text;

// ======================================================
// HEATING STATUS LEVEL
// ======================================================
IF GVL_STATE.G_Heating_Confidence > 0.8 THEN
    GVL_HMI.G_HMI_Heating_Status_Level := 0;
ELSIF GVL_STATE.G_Heating_Confidence > 0.5 THEN
    GVL_HMI.G_HMI_Heating_Status_Level := 1;
ELSE
    GVL_HMI.G_HMI_Heating_Status_Level := 2;
END_IF;

// ======================================================
// CASCADE SEMANTIC STATE
// ======================================================
GVL_HMI.G_HMI_Heating_Cascade_Available :=
    GVL_STATE.G_Heating_Cascade_Available;

GVL_HMI.G_HMI_Heating_Cascade_Degraded :=
    GVL_STATE.G_Heating_Cascade_Degraded;

GVL_HMI.G_HMI_Heating_Cascade_Partial_Capacity :=
    GVL_STATE.G_Heating_Cascade_Partial_Capacity;

GVL_HMI.G_HMI_Heating_Cascade_No_Flame :=
    GVL_STATE.G_Heating_Cascade_No_Flame;

GVL_HMI.G_HMI_Heating_Cascade_Transport_Degraded :=
    GVL_STATE.G_Heating_Cascade_Transport_Degraded;

GVL_HMI.G_HMI_Heating_Cascade_Ignition_Timeout :=
    GVL_STATE.G_Heating_Cascade_Ignition_Timeout;

GVL_HMI.G_HMI_Heating_Cascade_Active_Boilers :=
    GVL_STATE.G_Heating_Cascade_Active_Boilers;

GVL_HMI.G_HMI_Heating_Cascade_Available_Boilers :=
    GVL_STATE.G_Heating_Cascade_Available_Boilers;

// ======================================================
// OPENTHERM SEMANTIC STATE
// ======================================================
FOR L_i := 1 TO GVL_CONSTANTS.C_MAX_BOILERS DO

    GVL_HMI.G_HMI_Boiler_OT_Online[L_i] :=
        GVL_STATE.G_Boiler_OT_Online[L_i];

    GVL_HMI.G_HMI_Boiler_OT_Command_Ack[L_i] :=
        GVL_STATE.G_Boiler_OT_Command_Ack[L_i];

    GVL_HMI.G_HMI_Boiler_OT_Command_Timeout[L_i] :=
        GVL_STATE.G_Boiler_OT_Command_Timeout[L_i];

    GVL_HMI.G_HMI_Boiler_OT_Heartbeat_Timeout[L_i] :=
        GVL_STATE.G_Boiler_OT_Heartbeat_Timeout[L_i];

    GVL_HMI.G_HMI_Boiler_OT_Adapter_Error[L_i] :=
        GVL_STATE.G_Boiler_OT_Adapter_Error[L_i];

    GVL_HMI.G_HMI_Boiler_OT_Heartbeat_Age_MS[L_i] :=
        GVL_STATE.G_Boiler_OT_Heartbeat_Age_MS[L_i];

    GVL_HMI.G_HMI_Boiler_OT_Command_Age_MS[L_i] :=
        GVL_STATE.G_Boiler_OT_Command_Age_MS[L_i];

    GVL_HMI.G_HMI_Boiler_OT_Adapter_State[L_i] :=
        GVL_STATE.G_Boiler_OT_Adapter_State[L_i];

    GVL_HMI.G_HMI_Boiler_OT_Error_State[L_i] :=
        GVL_STATE.G_Boiler_OT_Error_State[L_i];

END_FOR;

// ======================================================
// PREDICTIVE FLAGS
// ======================================================
FOR L_i := 1 TO GVL_CONSTANTS.C_MAX_MANIFOLDS DO
    GVL_HMI.G_HMI_Heating_Predictive_Pressure_Drop[L_i] :=
        GVL_STATE.G_Predictive_Pump_Pressure_Drop[L_i];

    GVL_HMI.G_HMI_Heating_Predictive_Current_Rise[L_i] :=
        GVL_STATE.G_Predictive_Pump_Current_Rise[L_i];
END_FOR;

END_PROGRAM

(* ---- PRG_Modbus_RTU_Bridge.st ---- *)
PROGRAM PRG_Modbus_RTU_Bridge
VAR
    L_i : INT;
END_VAR

// ======================================================
// MODBUS RTU BRIDGE
// ======================================================
// This PRG transfers requests from the project runtime
// into the RTU bridge contract and applies confirmed responses.
//
// A concrete CODESYS Modbus RTU implementation must:
//   1. Observe G_Request_*
//   2. Execute physical RS485 transaction
//   3. Fill G_Response_*
//
// Safety:
//   - No response is generated internally.
//   - No fake Done is allowed.
// ======================================================

IF NOT GVL_MODBUS_RTU_BRIDGE.G_Bridge_Enabled THEN
    RETURN;
END_IF;

// ======================================================
// EXPORT FIRST ACTIVE REQUEST
// ======================================================
GVL_MODBUS_RTU_BRIDGE.G_Request_Valid := FALSE;

FOR L_i := 1 TO 16 DO

    IF GVL_MODBUS_MASTER.G_Request[L_i].Enable THEN

        GVL_MODBUS_RTU_BRIDGE.G_Request_Valid := TRUE;
        GVL_MODBUS_RTU_BRIDGE.G_Request_Index := L_i;
        GVL_MODBUS_RTU_BRIDGE.G_Request_Slave_ID :=
            GVL_MODBUS_MASTER.G_Request[L_i].Slave_ID;

        GVL_MODBUS_RTU_BRIDGE.G_Request_Function_Code :=
            GVL_MODBUS_MASTER.G_Request[L_i].Function_Code;

        GVL_MODBUS_RTU_BRIDGE.G_Request_Start_Register :=
            GVL_MODBUS_MASTER.G_Request[L_i].Start_Register;

        GVL_MODBUS_RTU_BRIDGE.G_Request_Register_Count :=
            GVL_MODBUS_MASTER.G_Request[L_i].Register_Count;

        GVL_MODBUS_RTU_BRIDGE.G_Request_Write_Value :=
            GVL_MODBUS_MASTER.G_Request[L_i].Write_Value;

        GVL_MODBUS_RTU_BRIDGE.G_Request_Sequence :=
            GVL_MODBUS_MASTER.G_Request[L_i].Sequence;

        GVL_MODBUS_RTU_BRIDGE.G_Request_Timeout_MS :=
            GVL_MODBUS_MASTER.G_Request[L_i].Timeout_MS;

        EXIT;
    END_IF;

END_FOR;

// ======================================================
// APPLY CONFIRMED RESPONSE
// ======================================================
IF GVL_MODBUS_RTU_BRIDGE.G_Response_Done OR
   GVL_MODBUS_RTU_BRIDGE.G_Response_Error THEN

    L_i := GVL_MODBUS_RTU_BRIDGE.G_Request_Index;

    IF (L_i >= 1) AND (L_i <= 16) THEN

        GVL_MODBUS_MASTER.G_Response[L_i].Busy :=
            GVL_MODBUS_RTU_BRIDGE.G_Response_Busy;

        GVL_MODBUS_MASTER.G_Response[L_i].Done :=
            GVL_MODBUS_RTU_BRIDGE.G_Response_Done;

        GVL_MODBUS_MASTER.G_Response[L_i].Error :=
            GVL_MODBUS_RTU_BRIDGE.G_Response_Error;

        GVL_MODBUS_MASTER.G_Response[L_i].Error_Code :=
            GVL_MODBUS_RTU_BRIDGE.G_Response_Error_Code;

        GVL_MODBUS_MASTER.G_Response[L_i].Read_Value :=
            GVL_MODBUS_RTU_BRIDGE.G_Response_Value;

        GVL_MODBUS_MASTER.G_Response[L_i].Last_Sequence :=
            GVL_MODBUS_RTU_BRIDGE.G_Response_Sequence;

        GVL_MODBUS_MASTER.G_Response[L_i].Last_Update_MS :=
            GVL_MODBUS_RTU_BRIDGE.G_Response_Update_MS;

    END_IF;

END_IF;

END_PROGRAM

(* ---- PRG_Modbus_RTU_SysCom_Transport.st ---- *)
PROGRAM PRG_Modbus_RTU_SysCom_Transport
VAR
    FB_SysCom_Transport : FB_Modbus_RTU_SysCom_Transport;
END_VAR

// ======================================================
// MODBUS RTU SYSCOM TRANSPORT EXECUTION
// ======================================================
// Byte-level transport boundary execution.
// ======================================================

FB_SysCom_Transport(
    VI_Enable := GVL_CONFIG.G_OpenTherm_Enabled,
    VI_System_Time_MS := GVL_STATUS.G_System_Time_MS
);

END_PROGRAM

(* ---- PRG_PLC_Arbitration.st ---- *)
PROGRAM PRG_PLC_Arbitration

// Update heartbeat
IF GVL_STATUS.G_Remote_PLC_Pulse THEN
    GVL_STATUS.G_Remote_PLC_Last_Seen_MS := GVL_TIME_SERVICE.G_Now_MS;
END_IF;

// Alive check (3s)
GVL_STATUS.G_Remote_PLC_Alive :=
    (GVL_TIME_SERVICE.G_Now_MS - GVL_STATUS.G_Remote_PLC_Last_Seen_MS) < 3000;

// Arbitration
IF NOT GVL_STATUS.G_Remote_PLC_Alive THEN
    GVL_STATUS.G_Is_Active_PLC := TRUE;
ELSE
    IF GVL_STATUS.G_Local_PLC_ID < GVL_STATUS.G_Active_PLC_ID THEN
        GVL_STATUS.G_Is_Active_PLC := TRUE;
    ELSE
        GVL_STATUS.G_Is_Active_PLC := FALSE;
    END_IF;
END_IF;

// >>> BULK_SYNC_ANCHOR: PRG_PLC_Arbitration <<<
END_PROGRAM

(* ---- PRG_System_Access_Maintenance.st ---- *)
PROGRAM PRG_System_Access_Maintenance
VAR
    fbLogEvent : FB_LogEvent;
    L_Dangerous_Action_Armed : BOOL;
    L_Dangerous_Action_Deadline_MS : UDINT;
    L_Maintenance_Apply_Intent : BOOL;
    L_User_Access_Denied_Prev : BOOL;
END_VAR

L_Maintenance_Apply_Intent := FALSE;

// Dangerous action request
IF GVL_COMMAND.CMD_Dangerous_Action_Request AND (GVL_COMMAND.CMD_User_Access_Level >= 2) THEN
    IF NOT L_Dangerous_Action_Armed THEN
        fbLogEvent(
            VI_Event_Type := 8,
            VI_Timestamp := GVL_TIME_SERVICE.G_Now_MS,
            VI_Param1 := TO_UDINT(GVL_COMMAND.CMD_User_Access_Level),
            VI_Param2 := 1
        );
    END_IF;

    L_Dangerous_Action_Armed := TRUE;
    L_Dangerous_Action_Deadline_MS := GVL_TIME_SERVICE.G_Now_MS + 15000;

    GVL_STATUS.G_Diagnostics.Dangerous_Action_Pending_Confirm := TRUE;
    GVL_STATUS.G_Diagnostics.Dangerous_Action_Confirm_Deadline_MS := L_Dangerous_Action_Deadline_MS;
    GVL_STATUS.G_Diagnostics.Dangerous_Action_Confirm_Text := 'Подтвердите опасное действие в течение 15 секунд';
END_IF;

// Timeout
IF L_Dangerous_Action_Armed AND (GVL_TIME_SERVICE.G_Now_MS > L_Dangerous_Action_Deadline_MS) THEN
    L_Dangerous_Action_Armed := FALSE;
    GVL_STATUS.G_Diagnostics.Dangerous_Action_Pending_Confirm := FALSE;
    GVL_STATUS.G_Diagnostics.Dangerous_Action_Confirm_Text := 'Окно подтверждения истекло';
END_IF;

// Confirm
IF GVL_COMMAND.CMD_Dangerous_Action_Confirm AND
   L_Dangerous_Action_Armed AND
   (GVL_COMMAND.CMD_User_Access_Level >= 2) THEN

    L_Maintenance_Apply_Intent := TRUE;

    fbLogEvent(
        VI_Event_Type := 9,
        VI_Timestamp := GVL_TIME_SERVICE.G_Now_MS,
        VI_Param1 := TO_UDINT(GVL_COMMAND.CMD_User_Access_Level),
        VI_Param2 := 1
    );

    L_Dangerous_Action_Armed := FALSE;
    GVL_STATUS.G_Diagnostics.Dangerous_Action_Pending_Confirm := FALSE;
    GVL_STATUS.G_Diagnostics.Dangerous_Action_Confirm_Text := 'Опасное действие подтверждено оператором';
END_IF;

// Apply maintenance
IF L_Maintenance_Apply_Intent THEN
    GVL_CONFIG.G_DHW_Heating_Pump_In_Service := GVL_COMMAND.CMD_Set_DHW_Heating_Pump_In_Service;
    GVL_CONFIG.G_DHW_Circ_Pump_In_Service := GVL_COMMAND.CMD_Set_DHW_Circ_Pump_In_Service;
END_IF;

// Access enforcement
GVL_STATUS.G_Diagnostics.User_Access_Level_Active := GVL_COMMAND.CMD_User_Access_Level;
GVL_STATUS.G_Diagnostics.User_Access_Denied := FALSE;

IF GVL_COMMAND.CMD_Dangerous_Action_Request OR GVL_COMMAND.CMD_Dangerous_Action_Confirm THEN
    IF GVL_COMMAND.CMD_User_Access_Level < 2 THEN
        IF NOT L_User_Access_Denied_Prev THEN
            fbLogEvent(
                VI_Event_Type := 10,
                VI_Timestamp := GVL_TIME_SERVICE.G_Now_MS,
                VI_Param1 := TO_UDINT(GVL_COMMAND.CMD_User_Access_Level),
                VI_Param2 := 2
            );
        END_IF;

        GVL_STATUS.G_Diagnostics.User_Access_Denied := TRUE;
        GVL_STATUS.G_Diagnostics.Operator_Action_Blocked := TRUE;
    END_IF;
END_IF;

L_User_Access_Denied_Prev := GVL_STATUS.G_Diagnostics.User_Access_Denied;

END_PROGRAM

(* ---- PRG_System_Diagnostics.st ---- *)
PROGRAM PRG_System_Diagnostics
VAR
    fbSystemDiagnostics : FB_System_Diagnostics;
    fbStateTraceLog : FB_State_Trace_Log;
    fbAdapt : FB_Behavior_Adapt;

    L_Pumps_4 : ARRAY[1..4] OF BOOL;
    L_i : INT;
    L_Last_State_Trace_MS : UDINT;

    L_Hum : REAL;
    L_PrevHum : REAL;
    L_DeltaHum : REAL;
    L_Confidence : REAL;
END_VAR

FOR L_i := 1 TO 4 DO
    L_Pumps_4[L_i] := GVL_HEATING_OUTPUT.DO_Manifold_Pumps[L_i];
END_FOR;

fbSystemDiagnostics();

fbStateTraceLog(
    VI_System_Time := GVL_TIME_SERVICE.G_Now_MS,
    VI_Gas_Alarm := GVL_ALARM.G_Gas_Alarm_Active,
    VI_Leak_Alarm := GVL_ALARM.G_Flood_Alarm_Active,
    VI_Pumps := L_Pumps_4,
    VO_Last_Change_Time => L_Last_State_Trace_MS
);

FOR L_i := 1 TO GVL_CONSTANTS.C_MAX_ZONES DO

    L_Hum := 0.0;

    IF GVL_BEHAVIOR_ADAPT.G_Prev_Valid[L_i] THEN
        L_PrevHum := GVL_BEHAVIOR_ADAPT.G_Prev_Humidity[L_i];
    ELSE
        L_PrevHum := L_Hum;
    END_IF;

    L_DeltaHum := L_PrevHum - L_Hum;

    IF ABS(L_DeltaHum) < 0.5 THEN
        L_Confidence := 0.2;
    ELSE
        L_Confidence := 1.0;
    END_IF;

    IF GVL_INTENT_BEHAVIOR.I_Request_Ventilation_Boost THEN
        fbAdapt(
            iScenario := REASON_SCENARIO_VENT_BOOST,
            iSuccess := (L_DeltaHum > 5.0),
            iMeasuredValue := L_Hum,
            iZone := L_i,
            iConfidence := L_Confidence
        );
    END_IF;

    GVL_BEHAVIOR_ADAPT.G_Prev_Humidity[L_i] := L_Hum;
    GVL_BEHAVIOR_ADAPT.G_Prev_Valid[L_i] := TRUE;

END_FOR;

IF GVL_INTENT_BEHAVIOR.I_Request_Night_Mode THEN
    fbAdapt(
        iScenario := REASON_SCENARIO_NIGHT,
        iSuccess := TRUE,
        iMeasuredValue := 0.0,
        iZone := 0,
        iConfidence := 1.0
    );
END_IF;

END_PROGRAM

(* ---- PRG_User_Adapt_Control.st ---- *)
PROGRAM PRG_User_Adapt_Control
VAR
    fbTrace : FB_Trace_Write;
    L_Text : STRING(64);
END_VAR

IF GVL_INTENT_USER.I_Set_Adapt_Profile_Req THEN

    // block if safety active
    IF (GVL_SAFETY_SHUTDOWN.G_Safety_Mode <> NORMAL) OR GVL_SAFETY_RECOVERY.G_Recovery_Active THEN

        fbTrace(
            iLayer := TRACE_USER,
            iSource := SRC_USER,
            iReason := REASON_SAFETY,
            iValueBool := FALSE,
            iValueReal := 0.0,
            iText := 'Profile change blocked: SAFETY ACTIVE'
        );

    ELSE

        IF (GVL_INTENT_USER.I_Set_Adapt_Profile_Confirm)
           AND (GVL_INTENT_USER.I_User_Access_Level >= 2) THEN

            GVL_BEHAVIOR_ADAPT.G_Adapt_Profile :=
                GVL_INTENT_USER.I_Adapt_Profile_Value;

            IF GVL_INTENT_USER.I_Adapt_Profile_Value = ADAPT_PROFILE_STABLE THEN
                L_Text := 'Adapt profile: STABLE';
            ELSIF GVL_INTENT_USER.I_Adapt_Profile_Value = ADAPT_PROFILE_BALANCED THEN
                L_Text := 'Adapt profile: BALANCED';
            ELSE
                L_Text := 'Adapt profile: AGGRESSIVE';
            END_IF;

            fbTrace(
                iLayer := TRACE_USER,
                iSource := SRC_USER,
                iReason := REASON_USER_REQUEST,
                iValueBool := TRUE,
                iValueReal := TO_REAL(GVL_INTENT_USER.I_User_Access_Level),
                iText := L_Text
            );

        END_IF;

    END_IF;

    GVL_INTENT_USER.I_Set_Adapt_Profile_Req := FALSE;
    GVL_INTENT_USER.I_Set_Adapt_Profile_Confirm := FALSE;

END_IF;
END_PROGRAM

(* ---- PRG_Water.st ---- *)
PROGRAM PRG_Water
VAR
    fbProjection : FB_Water_Output_Projection;
    L_Zone_Enable : ARRAY[1..GVL_CONSTANTS.C_MAX_WATER_ZONES] OF BOOL;
    L_Valve_35_Close : BOOL;
    L_Valve_36_Close : BOOL;
    L_i : INT;
END_VAR

FOR L_i := 1 TO GVL_CONSTANTS.C_MAX_WATER_ZONES DO
    L_Zone_Enable[L_i] := FALSE;
END_FOR;

IF GVL_INTENT_SAFETY.I_Water_Selective_Recovery_Allowed THEN
    IF (GVL_INTENT_SAFETY.I_Water_Recovery_Target_Zone >= 1) AND (GVL_INTENT_SAFETY.I_Water_Recovery_Target_Zone <= GVL_CONSTANTS.C_MAX_WATER_ZONES) THEN
        L_Zone_Enable[GVL_INTENT_SAFETY.I_Water_Recovery_Target_Zone] := TRUE;
    END_IF;
END_IF;

L_Valve_35_Close := GVL_COMMAND_SHADOW.G_Close_Valve_35;
L_Valve_36_Close := GVL_COMMAND_SHADOW.G_Close_Valve_36;

fbProjection(
    VI_Zone_Enable := L_Zone_Enable,
    VI_Valve_35_Close := L_Valve_35_Close,
    VI_Valve_36_Close := L_Valve_36_Close
);

// >>> BULK_SYNC_ANCHOR: PRG_Water <<<
END_PROGRAM
